FUNCTION_BLOCK FB_ManualControl
VAR_INPUT
	bEnable : BOOL;
	stParam : ST_Parameters;
END_VAR
VAR_OUTPUT
	fVelocityFeedForwardControlOutput : LREAL;
END_VAR
VAR
	fbJoystick : FB_Joystick; 
	fbOpenLoopControl : FB_OpenLoopControl; 
END_VAR

fbJoystick(
	bEnable := bEnable,
	stParam := stParam,
	fNormalizedInput := VirtualControlBox.stVirtualInputs.fJoystickY,
);

fbOpenLoopControl(
	bEnable := bEnable,
	stParam := stParam,
	fInput_ms := fbJoystick.fOuput,
	fMaxValveFlow_lmin := Parameters.stParam.fMaxFlowCapacity,
	fNormalizedOutput => fVelocityFeedForwardControlOutput
);

END_FUNCTION_BLOCK

(* stored: Version 1.1.0.1, ProductVersion 3.1.4024.9
   POU FB_ManualControl: Id {1cb952f3-59ec-4dc1-98d9-dc6242ed003b}, SpecialFunc None *)
